PROGRAM LightBulbTimer
VAR
	ONS :	BOOL;
END_VAR

IO();
(*Delays the LED for 10 seconds to turn on *)
//LEDTimer.On_DelayLED  (IN	:=	LightBulb.StartSignal = TRUE,  PT	:=	T#10S, Q=> , ET => );
//LEDTimer.Off_DelayLED (IN	:=	LightBulb.StopSignal = TRUE, PT	:=	T#10S,	Q=>, ET=> );


IF Lightbulb.StartSignal AND ONS THEN
	
	Lightbulb.YellowLED		:=	TRUE;
	Lightbulb.StopSignal	:=	FALSE;
	
END_IF

IF Lightbulb.StopSignal AND ONS = FALSE THEN

	Lightbulb.YellowLED		:=	FALSE;	
	Lightbulb.StartSignal	:=	FALSE;

END_IF

END_PROGRAM

(* stored: Version 1.1.0.1, ProductVersion 3.1.4024.9
   POU LightBulbTimer: Id {52afcbb2-5cdb-4618-b2b1-8b2f14a911b6}, SpecialFunc None *)
